{attribute addProperty BoxType "EL6001-0000-0020"}
{attribute addProperty Id "StatusAT %I*Status_A3013EBE8Data_InAT %I*ARRAY[0..49] OF UINT100"}
{attribute addProperty CRC "4202882230"}
{attribute addProperty SizeInBites "864"}
{attribute addProperty SizeInBytes "108"}
TYPE COM_ext_inputs_4889F9FB :
STRUCT
	{attribute addProperty Name "Status"}
	Status AT %I* : Status_A3013EBE;
	{attribute addProperty Name "Data_In"}
	Data_In AT %I* : ARRAY[0..49] OF UINT;
END_STRUCT
END_TYPE

(* stored: Version 1.2.0.0, ProductVersion 3.1.4024.9
   DUT COM_ext_inputs_4889F9FB: Id {e9323615-4c19-4273-b4a2-f7fc7710d4f1} *)
